FUNCTION_BLOCK INTERNAL MemoryCleanupHelper

//FB_Exit must be implemented explicitly. If there is an implementation, then the
//method is called before the controller removes the code of the function block instance
//(implicit call). The return value is not evaluated.
METHOD FB_Exit: BOOL
VAR_INPUT
    bInCopyCode: BOOL;  // TRUE: the exit method is called in order to leave the instance which will be copied afterwards (online change).  
END_VAR
DynamicMemoryManager.CleanupMemory(TRUE);
END_METHOD

END_FUNCTION_BLOCK

(* stored: Version 1.1.0.1
   POU MemoryCleanupHelper: Id {7dc830f2-0958-4a4b-8a4a-b4858028b05f}, SpecialFunc None
   Method FB_Exit: Id {ab8a9fe6-b7e4-4631-afbd-30ad2c87a604} *)
